PROGRAM MAIN
VAR
END_VAR

END_PROGRAM

(* stored: Version 1.1.0.1
   POU MAIN: Id {a0390e4c-5c81-42ee-9909-4d93e224b592} *)
